PROGRAM MAIN
VAR
END_VAR

END_PROGRAM

(* stored: Version 1.1.0.1, ProductVersion 3.1.0.36
   POU MAIN: Id {de34fbd4-cb1a-44f9-9c2b-1c58b3649359} *)
